PROGRAM MAIN
VAR
	fbTestSuites : FB_Testsuites;
	fbTestSuite : FB_Testsuite;
	
	MyCalculator : MyCalculatorClass;
	bExecute: BOOL;
END_VAR

fbTestSuites();
fbTestSuites.M_Add(fbTestSuite);
fbTestSuite();

IF bExecute THEN
	// manual execute | override file path
	fbTestsuites.P_Options.sFilePathName:= 'C:\Test\CalculatorTests.xml';
	bExecute:= NOT fbTestsuites.M_Request(E_Base.Execute);
END_IF

CASE fbTestSuite.P_Testcase OF
	E_Testcase.Start:
		fbTestSuite.P_Assert.M_Equals_INT(2, MyCalculator.Divide(4,2), 'Divide method did not return correct qoutient');
		fbTestSuite.M_Testcase('CalculatorClassShouldDivideTwoValidNumbers',T#1S,'','',1);
			 
	1:
		fbTestSuite.P_Assert.M_Equals_INT(-1, MyCalculator.Divide(4,0), 'Divide METHOD did NOT reject 0 divisor');
		fbTestSuite.M_Testcase('CalculatorClassShouldProhibitADivideByZero',T#1S,'','',E_Testcase.Done);

	E_Testcase.Done:;	 
END_CASE

END_PROGRAM

(* stored: Version 1.1.0.1, ProductVersion 3.1.4024.12
   POU MAIN: Id {3b11b508-effe-484a-b35c-e70da4aed0e0}, SpecialFunc None *)
